Yaskawa INFORM job: DM_PRINT.JBI

/JOB
//NAME DM_PRINT
//POS
///NPOS 0,0,0,0,0,0
//INST
///DATE 2025/02/20 16:20
///COMM Generated using RoboDK
///ATTR SC,RW
///GROUP1 RB1
NOP
CALL JOB:DPRINT3D
CALL JOB:DPRINT3D2
CALL JOB:DPRINT3D3
CALL JOB:DPRINT3D4
CALL JOB:DPRINT3D5
CALL JOB:DPRINT3D6
CALL JOB:DPRINT3D7
CALL JOB:DPRINT3D8
CALL JOB:DPRINT3D9
CALL JOB:DPRINT3D10
CALL JOB:DPRINT3D11
CALL JOB:DPRINT3D12
CALL JOB:DPRINT3D13
CALL JOB:DPRINT3D14
CALL JOB:DPRINT3D15
CALL JOB:DPRINT3D16
CALL JOB:DPRINT3D17
CALL JOB:DPRINT3D18
END
